# EPICS alarm handler configuration: alh_files/mgnt_li21_lgps.alhConfig
GROUP NULL LGPS:LI21:MG01
$ALIAS LGPS
$GUIDANCE
LI21 LGPS magnets
   Group Name: LGPS:LI21:MG01
   Summary PV:  LGPS:LI21:MG01:STATSUMY
$END

BOTH AREAS
GROUP LGPS:LI21:MG01  LGPS:LI21:2
CHANNEL     LGPS:LI21:2           LGPS:LI21:2:STATMSG   -----
   $FORCEPV LGPS:LI21:2:STATMSGSV -DATL 1 0
